// Mitsubishi GX Works2 project: 240507_timechart10_양음변환2   PLC: Q03UDV

PROGRAM MAIN
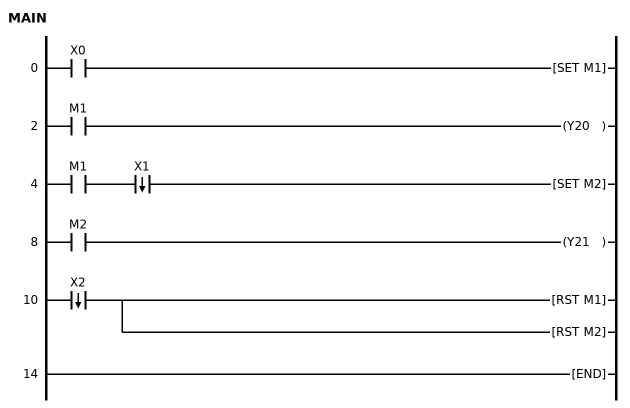
0     LD      X0
      SET     M1
2     LD      M1
      OUT     Y20
4     LD      M1
      ANDF    X1
      SET     M2
8     LD      M2
      OUT     Y21
10    LDF     X2
      RST     M1
      RST     M2
14    END
END_PROGRAM
